// TIA Portal project "AnaSuDepoTankıylaTesisIci4TankinDoldurmaUygulamasi" (V17)

(* hardware
DEVICE "S7-1200 station_1"  S7-1200 Station
   slot 0: "Rack_0"  S7-1200 Rack  Rack  V1.0
   slot 1: "PLC_1"  CPU 1214C DC/DC/DC  6ES7 214-1AG40-0XB0  V4.5
*)

// ===== PLC "PLC_1"  CPU 1214C DC/DC/DC =====

VAR_GLOBAL   // PLC tag table "Default tag table"
   "BOŞ SİNYALİ TANK 1" AT %I124.1 : Bool;
   "POMPA TANK 2" AT %Q124.2 : Bool;
   "POMPA TANK 3" AT %Q124.3 : Bool;
   "DOLU SİNYALİ TANK 1" AT %I124.0 : Bool;
   "POMPA TANK 1" AT %Q124.1 : Bool;
   "BOŞ SİNYALİ TANK 2" AT %I124.3 : Bool;
   "DOLU SİNYALİ TANK 2" AT %I124.2 : Bool;
   "BOŞ SİNYALİ TANK 3" AT %I124.5 : Bool;
   "DOLU SİNYALİ TANK 3" AT %I124.4 : Bool;
   "POMPA TANK 4" AT %Q124.4 : Bool;
   "BOŞ SİNYALİ TANK 4" AT %I124.7 : Bool;
   "DOLU SİNYALİ TANK 4" AT %I124.6 : Bool;
END_VAR

ORGANIZATION_BLOCK "Main"   // OB1, LAD, ProgramCycle
TITLE = "Main Program Sweep (Cycle)"
{ S7_Optimized_Access := 'TRUE' }
VERSION : 0.1
   VAR_INPUT
      Initial_Call : Bool;   // Initial call of this OB
      Remanence : Bool;   // =True, if remanent data are available
   END_VAR
BEGIN

REGION Network 1: POMPA 1
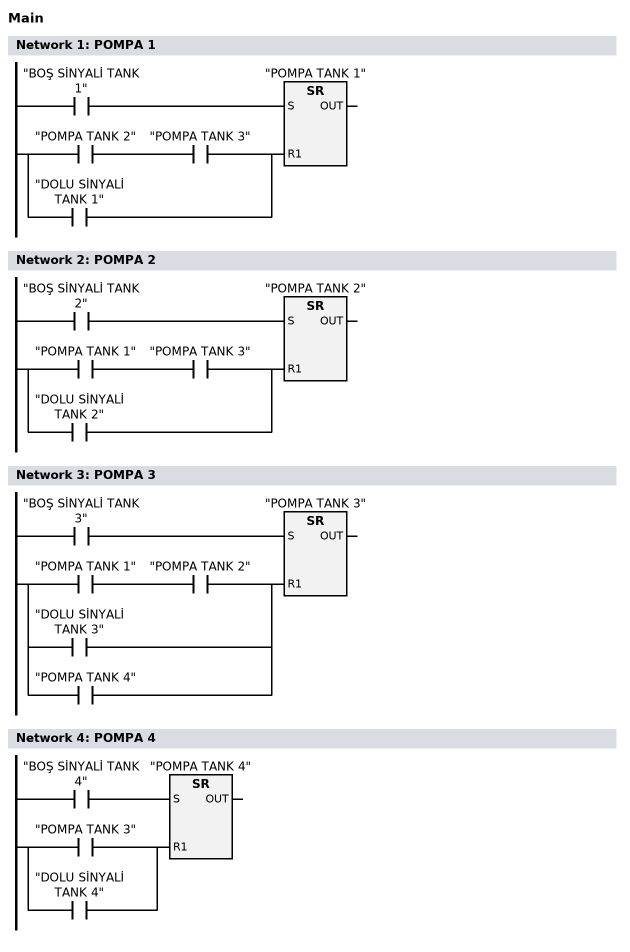
   RUNG wire#powerrail
      Contact( "BOŞ SİNYALİ TANK 1" )
      S_SR(operand := "POMPA TANK 1", r1 := wire#w1)
   END_RUNG
   RUNG wire#powerrail
      Contact( "POMPA TANK 2" )
      Contact( "POMPA TANK 3" )
   END_RUNG wire#w1
   RUNG wire#powerrail
      Contact( "DOLU SİNYALİ TANK 1" )
   END_RUNG wire#w1
   // the same network as SCL:
   IF "BOŞ SİNYALİ TANK 1" THEN
       "POMPA TANK 1" := TRUE;   // SR flip-flop
   END_IF;
   IF ("POMPA TANK 2" AND "POMPA TANK 3") OR "DOLU SİNYALİ TANK 1" THEN "POMPA TANK 1" := FALSE; END_IF;
END_REGION

REGION Network 2: POMPA 2
   RUNG wire#powerrail
      Contact( "BOŞ SİNYALİ TANK 2" )
      S_SR(operand := "POMPA TANK 2", r1 := wire#w1)
   END_RUNG
   RUNG wire#powerrail
      Contact( "POMPA TANK 1" )
      Contact( "POMPA TANK 3" )
   END_RUNG wire#w1
   RUNG wire#powerrail
      Contact( "DOLU SİNYALİ TANK 2" )
   END_RUNG wire#w1
   // the same network as SCL:
   IF "BOŞ SİNYALİ TANK 2" THEN
       "POMPA TANK 2" := TRUE;   // SR flip-flop
   END_IF;
   IF ("POMPA TANK 1" AND "POMPA TANK 3") OR "DOLU SİNYALİ TANK 2" THEN "POMPA TANK 2" := FALSE; END_IF;
END_REGION

REGION Network 3: POMPA 3
   RUNG wire#powerrail
      Contact( "BOŞ SİNYALİ TANK 3" )
      S_SR(operand := "POMPA TANK 3", r1 := wire#w1)
   END_RUNG
   RUNG wire#powerrail
      Contact( "POMPA TANK 1" )
      Contact( "POMPA TANK 2" )
   END_RUNG wire#w1
   RUNG wire#powerrail
      Contact( "DOLU SİNYALİ TANK 3" )
   END_RUNG wire#w1
   RUNG wire#powerrail
      Contact( "POMPA TANK 4" )
   END_RUNG wire#w1
   // the same network as SCL:
   IF "BOŞ SİNYALİ TANK 3" THEN
       "POMPA TANK 3" := TRUE;   // SR flip-flop
   END_IF;
   IF ("POMPA TANK 1" AND "POMPA TANK 2") OR "DOLU SİNYALİ TANK 3" OR "POMPA TANK 4" THEN
       "POMPA TANK 3" := FALSE;
   END_IF;
END_REGION

REGION Network 4: POMPA 4
   RUNG wire#powerrail
      Contact( "BOŞ SİNYALİ TANK 4" )
      S_SR(operand := "POMPA TANK 4", r1 := wire#w1)
   END_RUNG
   RUNG wire#powerrail
      Contact( "POMPA TANK 3" )
   END_RUNG wire#w1
   RUNG wire#powerrail
      Contact( "DOLU SİNYALİ TANK 4" )
   END_RUNG wire#w1
   // the same network as SCL:
   IF "BOŞ SİNYALİ TANK 4" THEN
       "POMPA TANK 4" := TRUE;   // SR flip-flop
   END_IF;
   IF "POMPA TANK 3" OR "DOLU SİNYALİ TANK 4" THEN "POMPA TANK 4" := FALSE; END_IF;
END_REGION
END_ORGANIZATION_BLOCK